FUNCTION_BLOCK Ave 
VAR_INPUT
END_VAR
VAR_OUTPUT
END_VAR
VAR
END_VAR

END_FUNCTION_BLOCK

(* stored: Version 1.1.0.1, ProductVersion 3.1.4024.12
   POU Ave: Id {b2def78c-68c0-4b6a-bb70-3ca08034a32e}, SpecialFunc None *)
